// TwinCAT 3 PLC project couple_demo_plc
// ProgramVersion: 3.1.4023.0
// CompilerDefines: VISU_USEWSTRING
// libraries:
//   Tc2_MC2, * (Beckhoff Automation GmbH)
//   Tc2_Standard, * (Beckhoff Automation GmbH)
//   Tc2_System, * (Beckhoff Automation GmbH)
//   Tc3_Module, * (Beckhoff Automation GmbH)
//   VisuDialogs, * (System)
//   VisuSymbols,3.5.10.0,System
// project tree:
//   / GlobalTextList.TcGTLO, PlcTask.TcTTO, VISU_TASK.TcTTO, 视图管理器.TcVMO (not stored)
//   POUs/couple/ master.TcPOU, slave.TcPOU, couple.TcPOU
//   POUs/ MAIN.TcPOU
//   VISUs/ coupleAxis.TcVIS (not stored)
// real-time tasks:
//   TASK PlcTask: cycle T#10ms, priority 20, ADS port 350
//   TASK VISU_TASK: cycle T#200000us, priority 30, ADS port 351
// motion (NC):
//   TASK NC-Task 1 SAF: cycle T#2ms, priority 4, ADS port 501
//   TASK NC-Task 1 SVB: cycle T#10ms, priority 8, ADS port 511
//   AXIS master (id 1)
//     OtherSettings: AllowMotionCmdToSlave=true
//     encoder EncType=1
//       EncPara: ScaleFactorNumerator=10, ScaleFactorDenominator=1048576
//     drive DrvType=5
//       Analog: TorqueSetpointScale=10, ScaleFactorActTorque=0.1
//       TimeComp: TaskDelayCycles=1
//     controller CtrType=1
//       CtrPara: PriorControlFactor=1
//         Observer: BandWidth=20
//   AXIS slave (id 2)
//     OtherSettings: AllowMotionCmdToSlave=true
//     encoder EncType=1
//       EncPara: ScaleFactorNumerator=10, ScaleFactorDenominator=1048576
//     drive DrvType=5
//       Analog: TorqueSetpointScale=10, ScaleFactorActTorque=0.1
//       TimeComp: TaskDelayCycles=1
//     controller CtrType=1
//       CtrPara: PriorControlFactor=1
//         Observer: BandWidth=20
// variable links:
//   couple_demo_plc/couple_demo_plc Instance <-> NC-Task 1 SAF/Axes/master
//     PlcTask Inputs/master.axis.NcToPlc <-> Outputs/ToPlc
//     PlcTask Outputs/master.axis.PlcToNc <-> Inputs/FromPlc
//   couple_demo_plc/couple_demo_plc Instance <-> NC-Task 1 SAF/Axes/slave
//     PlcTask Inputs/slave.axis.NcToPlc <-> Outputs/ToPlc
//     PlcTask Outputs/slave.axis.PlcToNc <-> Inputs/FromPlc

CONFIGURATION couple_demo_plc
    RESOURCE PLC ON TwinCAT3
        TASK PlcTask(INTERVAL := T#10ms, PRIORITY := 20);
        TASK VISU_TASK(INTERVAL := T#200000us, PRIORITY := 30);
        PROGRAM MAIN WITH PlcTask : MAIN;
        PROGRAM VisuElems_Visu_Prg WITH VISU_TASK : VisuElems.Visu_Prg;
    END_RESOURCE
END_CONFIGURATION

// ---- POUs/MAIN.TcPOU
PROGRAM MAIN
VAR
END_VAR

master.dummyAction();
slave.dummyAction();

couple.checkGearIn();
couple.checkGearOut();

master.checkPower();
slave.checkPower();

master.checkSetPoint();
slave.checkSetPoint();


master.checkMoving();
master.checkRelMove();

master.checkReset();
master.checkStop();
master.checkGoHome();

END_PROGRAM

// ---- POUs/couple/master.TcPOU
PROGRAM master
VAR
	axis: AXIS_REF;
	
	mcPower: MC_Power;
	shouldPowerOn: BOOL;
	isMotorReady: BOOL;
	
	mcSetPosition: MC_SetPosition;
	shouldSetZero: BOOL;
	
	mcJog: MC_Jog;
	shouldJog: BOOL;
	jogDirection: BOOL;
	
	mcMoveRelative: MC_MoveRelative;
	shouldMoveRel: BOOL;
	
	mcStop: MC_Stop;
	shouldStop:BOOL;
	
	mcReset: MC_Reset;
	shouldReset: BOOL;
	
	mcHome: MC_Home;
	shouldGoHome: BOOL;
	homeTrigger: BOOL;
END_VAR

METHOD checkGoHome : BOOL
VAR_INPUT
END_VAR
mcHome(
	Axis:= axis, 
	Execute:= shouldGoHome, 
	Position:= 0, 
	bCalibrationCam:= homeTrigger
);
END_METHOD

METHOD checkMoving : BOOL
VAR_STAT
END_VAR
IF isMotorReady THEN
	IF shouldJog THEN
		IF jogDirection THEN
		mcJog(
			Axis:= axis, 
			JogForward:= TRUE, 
			JogBackwards:= FALSE,
			Velocity:= 50);
		ELSE
			mcJog(
				Axis:= axis, 
				JogForward:= FALSE, 
				JogBackwards:= TRUE,
				Velocity:= 50);
		END_IF
	END_IF
END_IF
END_METHOD

METHOD checkPower : BOOL
VAR_INPUT
END_VAR
VAR
END_VAR
mcPower(
	Axis:= axis, 
	Enable:= shouldPowerOn, 
	Enable_Positive:= TRUE, 
	Enable_Negative:= TRUE,
	Status=> isMotorReady
);
END_METHOD

METHOD checkRelMove : BOOL
VAR_STAT
END_VAR
IF isMotorReady THEN
	mcMoveRelative(
		Axis:= axis, 
		Execute:= shouldMoveRel, 
		Distance:= 2000, 
		Velocity:= 50);
END_IF;
END_METHOD

METHOD checkReset : BOOL
IF isMotorReady THEN
	mcReset(
		Axis:= axis, 
		Execute:= shouldReset);
END_IF
END_METHOD

ACTION checkSetPoint:
mcSetPosition(
	Axis:= axis, 
	Execute:= shouldSetZero,
	Position := 0);
END_ACTION

METHOD checkStop : BOOL
VAR

END_VAR
IF isMotorReady THEN
	mcStop(
		Axis:= axis, 
		Execute:= shouldStop);
END_IF
END_METHOD

ACTION dummyAction:

END_ACTION

END_PROGRAM

// ---- POUs/couple/slave.TcPOU
PROGRAM slave
VAR
	axis: AXIS_REF;
	
	mcPower: MC_Power;
	shouldPowerOn: BOOL;
	isMotorReady: BOOL;
	
	mcSetPosition: MC_SetPosition;
	shouldSetZero: BOOL;
END_VAR

METHOD checkPower : BOOL
VAR_INPUT
END_VAR
mcPower(
	Axis:= axis, 
	Enable:= shouldPowerOn, 
	Enable_Positive:= TRUE, 
	Enable_Negative:= TRUE,
	Status=> isMotorReady
);
END_METHOD

ACTION checkSetPoint:
mcSetPosition(
	Axis:= axis, 
	Execute:= shouldSetZero,
	Position := 0);
END_ACTION

ACTION dummyAction:

END_ACTION

END_PROGRAM

// ---- POUs/couple/couple.TcPOU
PROGRAM couple
VAR
	mcGearIn: MC_GearIn;
	shouldGearIn: BOOL;
	
	mcGearOut: MC_GearOut;
	shouldGearOut: BOOL;
END_VAR

METHOD checkGearIn : BOOL
VAR_INPUT
END_VAR
mcGearIn(
	Master:= master.axis, 
	Slave:= slave.axis, 
	Execute:= shouldGearIn, 
	RatioNumerator:= 1, // 从轴速度
	RatioDenominator:= 1, // 主轴速度
	Acceleration:= , 
	Deceleration:= , 
	Jerk:= , 
	BufferMode:= , 
	Options:= , 
	InGear=> , 
	Busy=> , 
	Active=> , 
	CommandAborted=> , 
	Error=> , 
	ErrorID=> );
END_METHOD

METHOD checkGearOut : BOOL
VAR_INPUT
END_VAR
mcGearOut(
	Slave:= slave.axis, 
	Execute:= shouldGearOut, 
	Options:= , 
	Done=> , 
	Busy=> , 
	Error=> , 
	ErrorID=> );
END_METHOD

END_PROGRAM

// ---- GlobalTextList.TcGTLO
TEXTLIST GlobalTextList
  874 = 'axis1 %.2f'
  527 = 'axis1 set to zero'
  741 = 'axis1: %.2f'
  575 = 'axis1: .2f%'
  182 = 'axis2 set to zero'
  512 = 'axis2: %.2f'
  787 = 'gear in'
  963 = 'gear out'
  623 = 'home'
  830 = 'home trigger'
  341 = 'jog'
  111 = 'master set to zero'
  801 = 'master: %.2f'
  638 = 'moveRelative'
  205 = 'reset'
  673 = 'slave: %.2f'
  806 = 'slaveset to zero'
  186 = 'stop'
  526 = '只能静态耦合，动态解耦'
  456 = '电源'
  717 = '轴1上电'
  113 = '轴1电源'
END_TEXTLIST
